// TIA Portal V16 export
// export: Created 2023-03-29T11:03:36.8796163Z, ExportSetting WithDefaults, DisplayName Totally Integrated Automation Portal, DisplayVersion V16 Update 6, DisplayName TIA Portal Version Control Interface, DisplayVersion V16 Update 2, DisplayName TIA Portal Openness, DisplayVersion V16 Update 6, DisplayName STEP 7 Professional, DisplayVersion V16 Update 6, DisplayName STEP 7 Safety, DisplayVersion V16, DisplayName WinCC Advanced, DisplayVersion V16 Update 6
FUNCTION_BLOCK "VLV02_POSITION_old"   // FB17, LAD
TITLE = Valve driver 02
{ S7_Optimized_Access := 'FALSE' }
AUTHOR : RTecmer
VERSION : 0.2
// Driver 0-100% position drives
// Slowo STATUSU Napedu
// STAT - Prawy Byte
// WIZ  - Lewy Byte
//  
//   -STAT wektor stanu zaworu
//     -bit 0- alarm                                  (sygnal do SCADA)
//     -bit 1- zawor otwarty                    (sygnal do SCADA)
//     -bit 2-sterowanie zdal=1 loc=0 (sygnal do SCADA)
//     -bit 3- zawor zamkniety               (sygnal do SCADA)
//     -bit 4-otwieranie reczne              (sygnal z SCADA)
//     -bit 5-zamykanie reczne              (sygnal z SCADA)
//     -bit 6-alarm reset                        (sygnal z SCADA
//     -bit 8-auto= 1man=0                  (sygnal z SCADA)
//   -SUPV 
//   -CLSD zawor zamkniety                    - wejscie
//   -OPND zawor otwarty                        - wejscie
//   -REMT sterowanie zdal=1 loc=0      - wejscie
//   -OPEN otwarcie                                  - wyjscie
//   -CLSE zamkniecie                              - wyjscie
//   - TIM1 czas otwierania  
//   - TIM2 czas zamykania
// stored: AutoNumber false, IsIECCheckEnabled false, SetENOAutomatically false, UDAEnableTagReadback false
   VAR_INPUT
      SetOpen_Percent { ExternalAccessible := 'False'; ExternalVisible := 'False'; ExternalWritable := 'False'} : Word;   // Zadany procent otwarcia
      VectorOut { ExternalAccessible := 'False'; ExternalVisible := 'False'; ExternalWritable := 'False'} : Word;   // Wektor otwarcia z nadajnika
      CLSD : Bool;   // Zamknięta
      OPND : Bool;   // Otwarta
      REMT : Bool;   // Sterowanie zdalne =1, remontowe=0
   END_VAR
   VAR_IN_OUT
      CLSE { ExternalAccessible := 'False'; ExternalVisible := 'False'; ExternalWritable := 'False'} : Bool;   // Wyjście zamykanie
      OPEN { ExternalAccessible := 'False'; ExternalVisible := 'False'; ExternalWritable := 'False'} : Bool;   // Wyjście Otwieranie
      WIZ : Byte;   // Wektor SCADA
      STAT : Byte;   // Wektor statusu napędu
      TMR1 : IEC_TIMER;   // Timer
   END_VAR
   VAR_TEMP
      SVMC : Bool;   // Automat na zamykanie
      SVMO : Bool;   // Automat na otwieranie
      man_Close : Bool;   // znacznik zamykania w trymie manual
      man_Open : Bool;   // znacznik otwierania w trybie manual
      instDiffOpen : Real;   // róznica kąta otwarcia zasuwy
      SP_Real : Real;   // Zadana wartość po konwersji
      PV_Real : Real;   // Vektor położeia po konwerski
      Diff_Real : Real;   // różnica po konwersji
      tmpError_Open : Bool;   // pomocniczy znacznik kontroli czasu jazdy na otwieranie
      tmpError_Close : Bool;   // pomocniczy znacznik kontroli czasu jazdy na zamykanie
   END_VAR
BEGIN

REGION Network 1
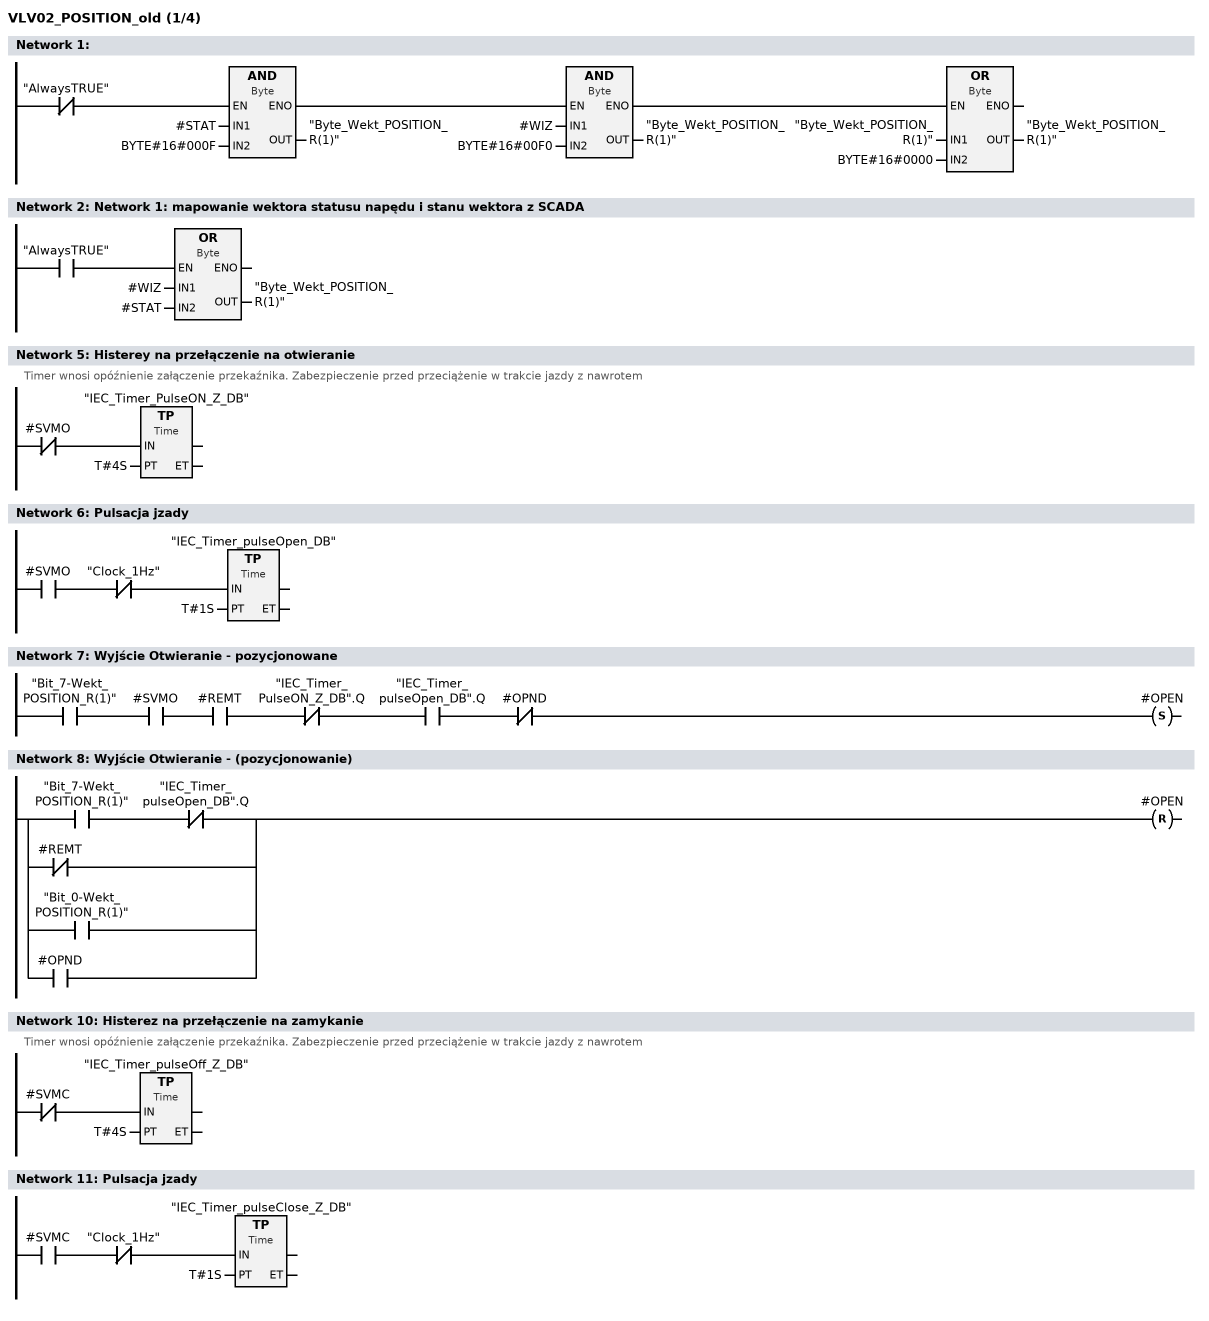
   IF NOT "AlwaysTRUE" THEN
       "Byte_Wekt_POSITION_R(1)" := #STAT AND BYTE#16#000F;
       "Byte_Wekt_POSITION_R(1)" := #WIZ AND BYTE#16#00F0;
       "Byte_Wekt_POSITION_R(1)" := "Byte_Wekt_POSITION_R(1)" OR BYTE#16#0000;
   END_IF;
END_REGION

REGION Network 2: Network 1: mapowanie wektora statusu napędu i stanu wektora z SCADA
   IF "AlwaysTRUE" THEN "Byte_Wekt_POSITION_R(1)" := #WIZ OR #STAT; END_IF;
END_REGION

REGION Network 3 (SCL): wyliczenie różnicy położenia
   //wyliczenie różnicy położenia
   REGION Konwersja zmiennych 
     // Konwersja do Real
     #SP_Real := INT_TO_REAL(#SetOpen_Percent);
     #PV_Real := INT_TO_REAL(#VectorOut);

   END_REGION

   #Diff_Real := (#SP_Real - #PV_Real);
   #instDiffOpen := #Diff_Real;
END_REGION

REGION Network 4 (SCL): Wyznaczenie wektora i jazda na otwierane


   //Strowanie na otwieranie 
   IF #REMT AND ("Bit_0-Wekt_POSITION_R(1)" = FALSE )THEN
     // Porównaj wartość różnicy do 1
     IF #instDiffOpen > 1.0 AND (#OPND = FALSE )AND ("Bit_0-Wekt_POSITION_R(1)" = TRUE) THEN
       // ustaw znacznik automatyczne otwieranie
       #SVMO := TRUE;
       // znacznik do kontroli czasu 
       #tmpError_Open := TRUE;
     ELSE
       #SVMO := FALSE;
       #tmpError_Open:= FALSE
       ;
     END_IF;

     ;
   END_IF;
END_REGION

REGION Network 5: Histerey na przełączenie na otwieranie
   // Timer wnosi opóźnienie załączenie przekaźnika. Zabezpieczenie przed przeciążenie w trakcie jazdy z nawrotem
   RUNG wire#powerrail
      I_Contact( #SVMO )
      { S7_Templates := "time_type := Time" } "IEC_Timer_PulseON_Z_DB".TP(pt := T#4S, et =>)
   END_RUNG
   // the same network as SCL:
   "IEC_Timer_PulseON_Z_DB".TP(IN := NOT #SVMO, PT := T#4S);
END_REGION

REGION Network 6: Pulsacja jzady
   RUNG wire#powerrail
      Contact( #SVMO )
      I_Contact( "Clock_1Hz" )
      { S7_Templates := "time_type := Time" } "IEC_Timer_pulseOpen_DB".TP(pt := T#1S, et =>)
   END_RUNG
   // the same network as SCL:
   "IEC_Timer_pulseOpen_DB".TP(IN := #SVMO AND NOT "Clock_1Hz", PT := T#1S);
END_REGION

REGION Network 7: Wyjście Otwieranie - pozycjonowane
   RUNG wire#powerrail
      Contact( "Bit_7-Wekt_POSITION_R(1)" )
      Contact( #SVMO )
      Contact( #REMT )
      I_Contact( "IEC_Timer_PulseON_Z_DB".Q )
      Contact( "IEC_Timer_pulseOpen_DB".Q )
      I_Contact( #OPND )
      S_Coil( #OPEN )
   END_RUNG
   // the same network as SCL:
   IF "Bit_7-Wekt_POSITION_R(1)" AND #SVMO AND #REMT AND NOT "IEC_Timer_PulseON_Z_DB".Q AND "IEC_Timer_pulseOpen_DB".Q AND NOT #OPND THEN
       #OPEN := TRUE;
   END_IF;
END_REGION

REGION Network 8: Wyjście Otwieranie - (pozycjonowanie)
   RUNG wire#powerrail
      Contact( "Bit_7-Wekt_POSITION_R(1)" )
      I_Contact( "IEC_Timer_pulseOpen_DB".Q )
      wire#w1
      R_Coil( #OPEN )
   END_RUNG
   RUNG wire#powerrail
      I_Contact( #REMT )
   END_RUNG wire#w1
   RUNG wire#powerrail
      Contact( "Bit_0-Wekt_POSITION_R(1)" )
   END_RUNG wire#w1
   RUNG wire#powerrail
      Contact( #OPND )
   END_RUNG wire#w1
   // the same network as SCL:
   IF ("Bit_7-Wekt_POSITION_R(1)" AND NOT "IEC_Timer_pulseOpen_DB".Q) OR NOT #REMT OR "Bit_0-Wekt_POSITION_R(1)" OR #OPND THEN
       #OPEN := FALSE;
   END_IF;
END_REGION

REGION Network 9 (SCL): Wyznaczenie wektora i jazda na zamykanie



   //Strowanie na zamykanie
   IF #REMT AND ("Bit_0-Wekt_POSITION_R(1)" = FALSE )THEN
     // Porównaj wartość różnicy do 1
     IF #instDiffOpen < -1.0 AND (#CLSD = FALSE) AND ("Bit_0-Wekt_POSITION_R(1)" = TRUE) THEN
       // ustaw znacznik automatyczne zamykanie
       #SVMC := TRUE;
       // znacznik kontroli czasu jazdy
       #tmpError_Close := TRUE;
     ELSE
       #SVMC := FALSE;
       #tmpError_Close:= FALSE
       ;
     END_IF;

     ;
   END_IF;
END_REGION

REGION Network 10: Histerez na przełączenie na zamykanie
   // Timer wnosi opóźnienie załączenie przekaźnika. Zabezpieczenie przed przeciążenie w trakcie jazdy z nawrotem
   RUNG wire#powerrail
      I_Contact( #SVMC )
      { S7_Templates := "time_type := Time" } "IEC_Timer_pulseOff_Z_DB".TP(pt := T#4S, et =>)
   END_RUNG
   // the same network as SCL:
   "IEC_Timer_pulseOff_Z_DB".TP(IN := NOT #SVMC, PT := T#4S);
END_REGION

REGION Network 11: Pulsacja jzady
   RUNG wire#powerrail
      Contact( #SVMC )
      I_Contact( "Clock_1Hz" )
      { S7_Templates := "time_type := Time" } "IEC_Timer_pulseClose_Z_DB".TP(pt := T#1S, et =>)
   END_RUNG
   // the same network as SCL:
   "IEC_Timer_pulseClose_Z_DB".TP(IN := #SVMC AND NOT "Clock_1Hz", PT := T#1S);
END_REGION

REGION Network 12: Wyjście zamykanie - pozycjonowane
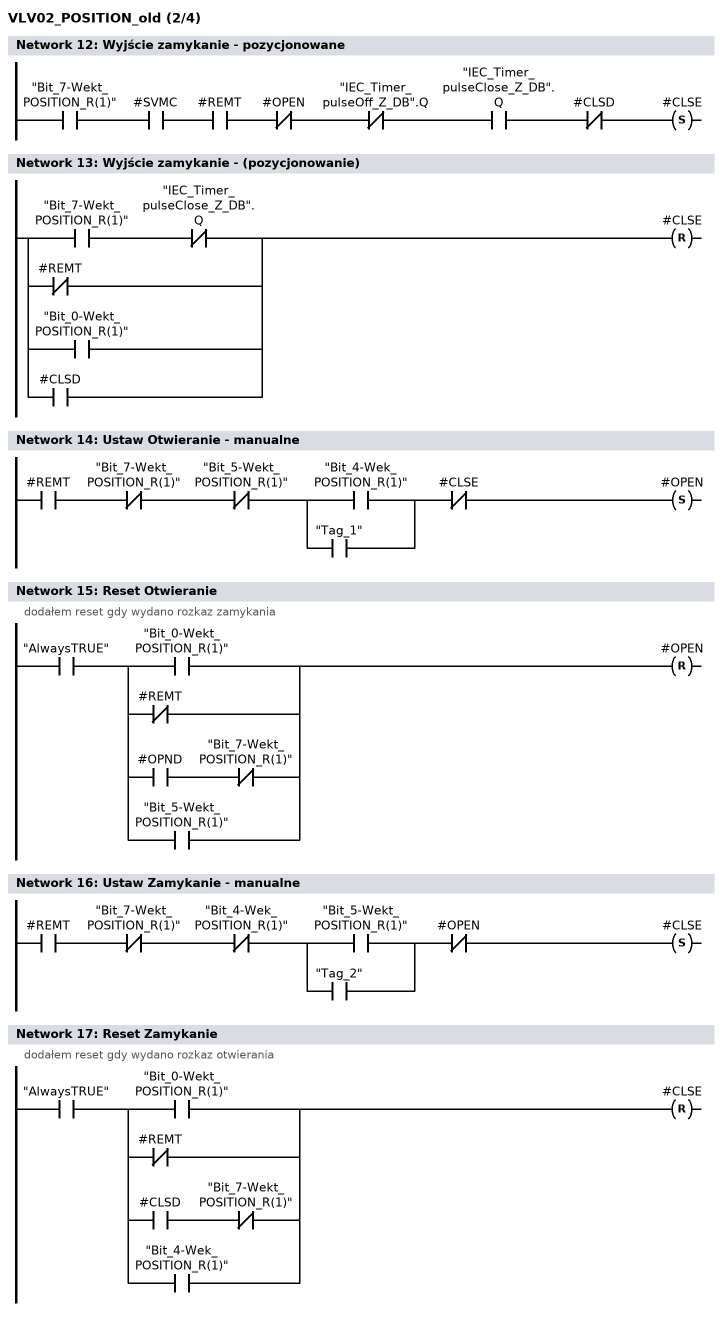
   RUNG wire#powerrail
      Contact( "Bit_7-Wekt_POSITION_R(1)" )
      Contact( #SVMC )
      Contact( #REMT )
      I_Contact( #OPEN )
      I_Contact( "IEC_Timer_pulseOff_Z_DB".Q )
      Contact( "IEC_Timer_pulseClose_Z_DB".Q )
      I_Contact( #CLSD )
      S_Coil( #CLSE )
   END_RUNG
   // the same network as SCL:
   IF "Bit_7-Wekt_POSITION_R(1)" AND #SVMC AND #REMT AND NOT #OPEN AND NOT "IEC_Timer_pulseOff_Z_DB".Q AND "IEC_Timer_pulseClose_Z_DB".Q AND NOT #CLSD THEN
       #CLSE := TRUE;
   END_IF;
END_REGION

REGION Network 13: Wyjście zamykanie - (pozycjonowanie)
   RUNG wire#powerrail
      Contact( "Bit_7-Wekt_POSITION_R(1)" )
      I_Contact( "IEC_Timer_pulseClose_Z_DB".Q )
      wire#w1
      R_Coil( #CLSE )
   END_RUNG
   RUNG wire#powerrail
      I_Contact( #REMT )
   END_RUNG wire#w1
   RUNG wire#powerrail
      Contact( "Bit_0-Wekt_POSITION_R(1)" )
   END_RUNG wire#w1
   RUNG wire#powerrail
      Contact( #CLSD )
   END_RUNG wire#w1
   // the same network as SCL:
   IF ("Bit_7-Wekt_POSITION_R(1)" AND NOT "IEC_Timer_pulseClose_Z_DB".Q) OR NOT #REMT OR "Bit_0-Wekt_POSITION_R(1)" OR #CLSD THEN
       #CLSE := FALSE;
   END_IF;
END_REGION

REGION Network 14: Ustaw Otwieranie - manualne
   RUNG wire#powerrail
      Contact( #REMT )
      I_Contact( "Bit_7-Wekt_POSITION_R(1)" )
      I_Contact( "Bit_5-Wekt_POSITION_R(1)" )
      wire#w1
      Contact( "Bit_4-Wek_POSITION_R(1)" )
      wire#w2
      I_Contact( #CLSE )
      S_Coil( #OPEN )
   END_RUNG
   RUNG wire#w1
      Contact( "Tag_1" )
   END_RUNG wire#w2
   // the same network as SCL:
   IF #REMT AND NOT "Bit_7-Wekt_POSITION_R(1)" AND NOT "Bit_5-Wekt_POSITION_R(1)" AND ("Bit_4-Wek_POSITION_R(1)" OR "Tag_1") AND NOT #CLSE THEN
       #OPEN := TRUE;
   END_IF;
END_REGION

REGION Network 15: Reset Otwieranie
   // dodałem reset gdy wydano rozkaz zamykania
   RUNG wire#powerrail
      Contact( "AlwaysTRUE" )
      wire#w1
      Contact( "Bit_0-Wekt_POSITION_R(1)" )
      wire#w2
      R_Coil( #OPEN )
   END_RUNG
   RUNG wire#w1
      I_Contact( #REMT )
   END_RUNG wire#w2
   RUNG wire#w1
      Contact( #OPND )
      I_Contact( "Bit_7-Wekt_POSITION_R(1)" )
   END_RUNG wire#w2
   RUNG wire#w1
      Contact( "Bit_5-Wekt_POSITION_R(1)" )
   END_RUNG wire#w2
   // the same network as SCL:
   IF "AlwaysTRUE" AND ("Bit_0-Wekt_POSITION_R(1)" OR NOT #REMT OR (#OPND AND NOT "Bit_7-Wekt_POSITION_R(1)") OR "Bit_5-Wekt_POSITION_R(1)") THEN
       #OPEN := FALSE;
   END_IF;
END_REGION

REGION Network 16: Ustaw Zamykanie - manualne
   RUNG wire#powerrail
      Contact( #REMT )
      I_Contact( "Bit_7-Wekt_POSITION_R(1)" )
      I_Contact( "Bit_4-Wek_POSITION_R(1)" )
      wire#w1
      Contact( "Bit_5-Wekt_POSITION_R(1)" )
      wire#w2
      I_Contact( #OPEN )
      S_Coil( #CLSE )
   END_RUNG
   RUNG wire#w1
      Contact( "Tag_2" )
   END_RUNG wire#w2
   // the same network as SCL:
   IF #REMT AND NOT "Bit_7-Wekt_POSITION_R(1)" AND NOT "Bit_4-Wek_POSITION_R(1)" AND ("Bit_5-Wekt_POSITION_R(1)" OR "Tag_2") AND NOT #OPEN THEN
       #CLSE := TRUE;
   END_IF;
END_REGION

REGION Network 17: Reset Zamykanie
   // dodałem reset gdy wydano rozkaz otwierania
   RUNG wire#powerrail
      Contact( "AlwaysTRUE" )
      wire#w1
      Contact( "Bit_0-Wekt_POSITION_R(1)" )
      wire#w2
      R_Coil( #CLSE )
   END_RUNG
   RUNG wire#w1
      I_Contact( #REMT )
   END_RUNG wire#w2
   RUNG wire#w1
      Contact( #CLSD )
      I_Contact( "Bit_7-Wekt_POSITION_R(1)" )
   END_RUNG wire#w2
   RUNG wire#w1
      Contact( "Bit_4-Wek_POSITION_R(1)" )
   END_RUNG wire#w2
   // the same network as SCL:
   IF "AlwaysTRUE" AND ("Bit_0-Wekt_POSITION_R(1)" OR NOT #REMT OR (#CLSD AND NOT "Bit_7-Wekt_POSITION_R(1)") OR "Bit_4-Wek_POSITION_R(1)") THEN
       #CLSE := FALSE;
   END_IF;
END_REGION

REGION Network 19: Kontrola awayjnego zlepienia styczników
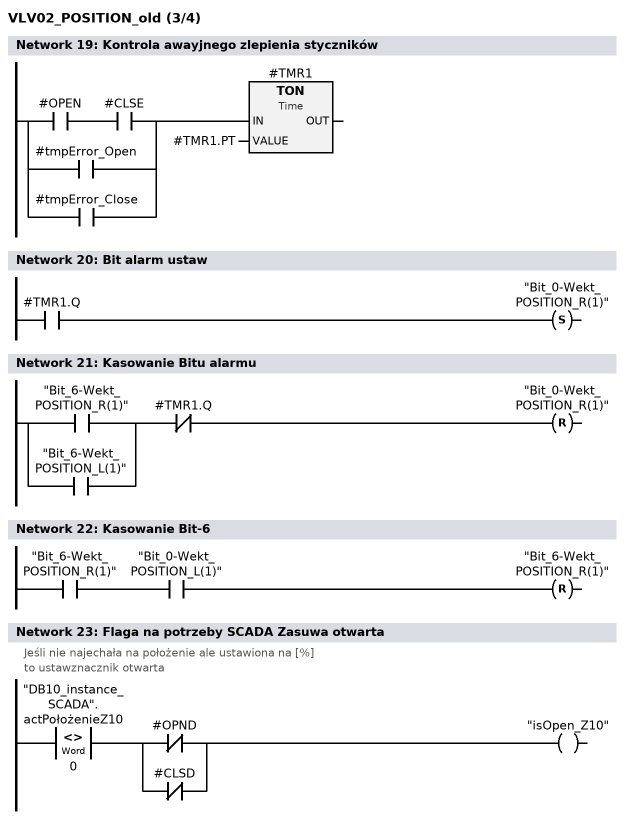
   #TMR1.TON(IN := (#OPEN AND #CLSE) OR #tmpError_Open OR #tmpError_Close, PT := #TMR1.PT);   // TON coil
END_REGION

REGION Network 20: Bit alarm ustaw
   RUNG wire#powerrail
      Contact( #TMR1.Q )
      S_Coil( "Bit_0-Wekt_POSITION_R(1)" )
   END_RUNG
   // the same network as SCL:
   IF #TMR1.Q THEN "Bit_0-Wekt_POSITION_R(1)" := TRUE; END_IF;
END_REGION

REGION Network 21: Kasowanie Bitu alarmu
   RUNG wire#powerrail
      Contact( "Bit_6-Wekt_POSITION_R(1)" )
      wire#w1
      I_Contact( #TMR1.Q )
      R_Coil( "Bit_0-Wekt_POSITION_R(1)" )
   END_RUNG
   RUNG wire#powerrail
      Contact( "Bit_6-Wekt_POSITION_L(1)" )
   END_RUNG wire#w1
   // the same network as SCL:
   IF ("Bit_6-Wekt_POSITION_R(1)" OR "Bit_6-Wekt_POSITION_L(1)") AND NOT #TMR1.Q THEN
       "Bit_0-Wekt_POSITION_R(1)" := FALSE;
   END_IF;
END_REGION

REGION Network 22: Kasowanie Bit-6
   RUNG wire#powerrail
      Contact( "Bit_6-Wekt_POSITION_R(1)" )
      Contact( "Bit_0-Wekt_POSITION_L(1)" )
      R_Coil( "Bit_6-Wekt_POSITION_R(1)" )
   END_RUNG
   // the same network as SCL:
   IF "Bit_6-Wekt_POSITION_R(1)" AND "Bit_0-Wekt_POSITION_L(1)" THEN
       "Bit_6-Wekt_POSITION_R(1)" := FALSE;
   END_IF;
END_REGION

REGION Network 23: Flaga na potrzeby SCADA Zasuwa otwarta
   // Jeśli nie najechała na położenie ale ustawiona na [%]
   // to ustawznacznik otwarta
   RUNG wire#powerrail
      { S7_Templates := "SrcType := Word" } NE_Contact(in1 := "DB10_instance_SCADA".actPołożenieZ10, in2 := 0)
      wire#w1
      I_Contact( #OPND )
      wire#w2
      Coil( "isOpen_Z10" )
   END_RUNG
   RUNG wire#w1
      I_Contact( #CLSD )
   END_RUNG wire#w2
   // the same network as SCL:
   "isOpen_Z10" := ("DB10_instance_SCADA".actPołożenieZ10 <> 0) AND (NOT #OPND OR NOT #CLSD);
END_REGION

REGION Network 24: Przepisanie Byte Wektora napędu
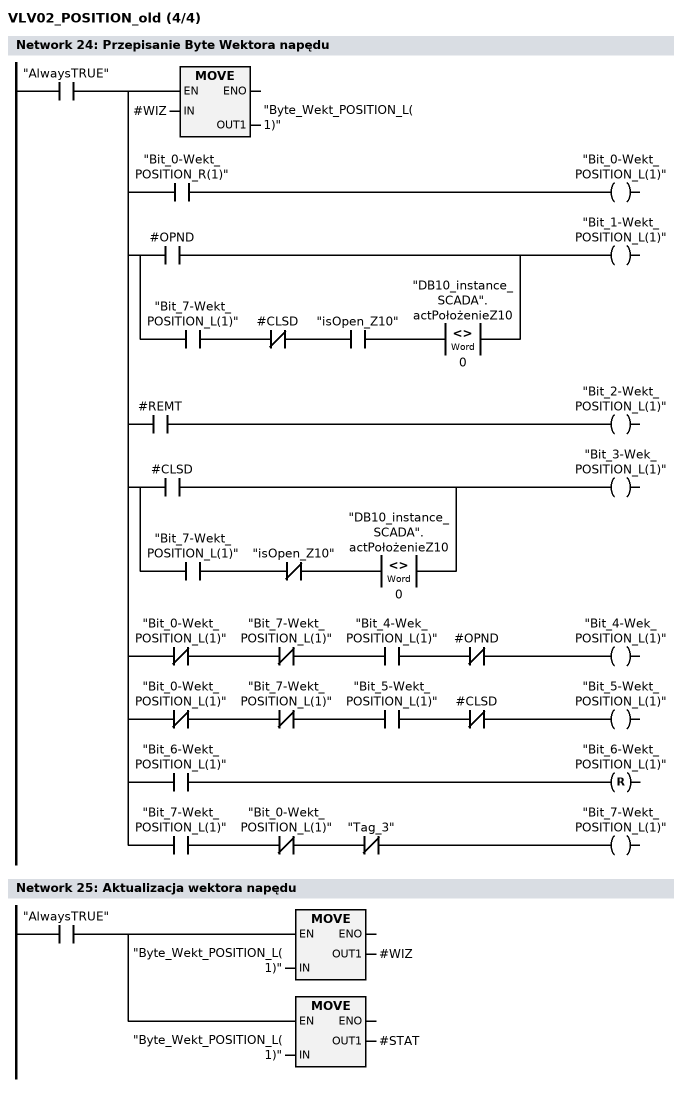
   RUNG wire#powerrail
      Contact( "AlwaysTRUE" )
      wire#w1
      { S7_GenerateENO := "TRUE" } Move(in := #WIZ, out1 => "Byte_Wekt_POSITION_L(1)")
   END_RUNG
   RUNG wire#w1
      Contact( "Bit_0-Wekt_POSITION_R(1)" )
      Coil( "Bit_0-Wekt_POSITION_L(1)" )
   END_RUNG
   RUNG wire#w1
      Contact( #OPND )
      wire#w2
      Coil( "Bit_1-Wekt_POSITION_L(1)" )
   END_RUNG
   RUNG wire#w1
      Contact( "Bit_7-Wekt_POSITION_L(1)" )
      I_Contact( #CLSD )
      Contact( "isOpen_Z10" )
      { S7_Templates := "SrcType := Word" } NE_Contact(in1 := "DB10_instance_SCADA".actPołożenieZ10, in2 := 0)
   END_RUNG wire#w2
   RUNG wire#w1
      Contact( #REMT )
      Coil( "Bit_2-Wekt_POSITION_L(1)" )
   END_RUNG
   RUNG wire#w1
      Contact( #CLSD )
      wire#w3
      Coil( "Bit_3-Wek_POSITION_L(1)" )
   END_RUNG
   RUNG wire#w1
      Contact( "Bit_7-Wekt_POSITION_L(1)" )
      I_Contact( "isOpen_Z10" )
      { S7_Templates := "SrcType := Word" } NE_Contact(in1 := "DB10_instance_SCADA".actPołożenieZ10, in2 := 0)
   END_RUNG wire#w3
   RUNG wire#w1
      I_Contact( "Bit_0-Wekt_POSITION_L(1)" )
      I_Contact( "Bit_7-Wekt_POSITION_L(1)" )
      Contact( "Bit_4-Wek_POSITION_L(1)" )
      I_Contact( #OPND )
      Coil( "Bit_4-Wek_POSITION_L(1)" )
   END_RUNG
   RUNG wire#w1
      I_Contact( "Bit_0-Wekt_POSITION_L(1)" )
      I_Contact( "Bit_7-Wekt_POSITION_L(1)" )
      Contact( "Bit_5-Wekt_POSITION_L(1)" )
      I_Contact( #CLSD )
      Coil( "Bit_5-Wekt_POSITION_L(1)" )
   END_RUNG
   RUNG wire#w1
      Contact( "Bit_6-Wekt_POSITION_L(1)" )
      R_Coil( "Bit_6-Wekt_POSITION_L(1)" )
   END_RUNG
   RUNG wire#w1
      Contact( "Bit_7-Wekt_POSITION_L(1)" )
      I_Contact( "Bit_0-Wekt_POSITION_L(1)" )
      I_Contact( "Tag_3" )
      Coil( "Bit_7-Wekt_POSITION_L(1)" )
   END_RUNG
   // the same network as SCL:
   IF "AlwaysTRUE" THEN "Byte_Wekt_POSITION_L(1)" := #WIZ; END_IF;
   "Bit_0-Wekt_POSITION_L(1)" := "AlwaysTRUE" AND "Bit_0-Wekt_POSITION_R(1)";
   "Bit_1-Wekt_POSITION_L(1)" := "AlwaysTRUE" AND (#OPND OR ("Bit_7-Wekt_POSITION_L(1)" AND NOT #CLSD AND "isOpen_Z10" AND ("DB10_instance_SCADA".actPołożenieZ10 <> 0)));
   "Bit_2-Wekt_POSITION_L(1)" := "AlwaysTRUE" AND #REMT;
   "Bit_3-Wek_POSITION_L(1)" := "AlwaysTRUE" AND (#CLSD OR ("Bit_7-Wekt_POSITION_L(1)" AND NOT "isOpen_Z10" AND ("DB10_instance_SCADA".actPołożenieZ10 <> 0)));
   "Bit_4-Wek_POSITION_L(1)" := "AlwaysTRUE" AND NOT "Bit_0-Wekt_POSITION_L(1)" AND NOT "Bit_7-Wekt_POSITION_L(1)" AND "Bit_4-Wek_POSITION_L(1)" AND NOT #OPND;
   "Bit_5-Wekt_POSITION_L(1)" := "AlwaysTRUE" AND NOT "Bit_0-Wekt_POSITION_L(1)" AND NOT "Bit_7-Wekt_POSITION_L(1)" AND "Bit_5-Wekt_POSITION_L(1)" AND NOT #CLSD;
   IF "AlwaysTRUE" AND "Bit_6-Wekt_POSITION_L(1)" THEN "Bit_6-Wekt_POSITION_L(1)" := FALSE; END_IF;
   "Bit_7-Wekt_POSITION_L(1)" := "AlwaysTRUE" AND "Bit_7-Wekt_POSITION_L(1)" AND NOT "Bit_0-Wekt_POSITION_L(1)" AND NOT "Tag_3";
END_REGION

REGION Network 25: Aktualizacja wektora napędu
   RUNG wire#powerrail
      Contact( "AlwaysTRUE" )
      wire#w1
      { S7_GenerateENO := "TRUE" } Move(in := "Byte_Wekt_POSITION_L(1)", out1 => #WIZ)
   END_RUNG
   RUNG wire#w1
      { S7_GenerateENO := "TRUE" } Move(in := "Byte_Wekt_POSITION_L(1)", out1 => #STAT)
   END_RUNG
   // the same network as SCL:
   IF "AlwaysTRUE" THEN
       #WIZ := "Byte_Wekt_POSITION_L(1)";
       #STAT := "Byte_Wekt_POSITION_L(1)";
   END_IF;
END_REGION
END_FUNCTION_BLOCK
